PROGRAM PRG_Com
VAR
END_VAR

(*Instanitate Serial port com function *) 
//ChemRIXS PTM_03 
K2S17_E5_CH2_fbSerialLineControl(
	Mode:= SERIALLINEMODE_EL6_22B,
	pComIn:= ADR(K2S17_E5_CH2_stComIn),
	pComOut:=ADR(K2S17_E5_CH2_stComOut),
	SizeComIn:= SIZEOF(K2S17_E5_CH2_stComOut),
	TxBuffer:= K2S17_E5_CH2_SerialTXBuffer,
	RxBuffer:= K2S17_E5_CH2_SerialRXBuffer,
	Error=> ,
	ErrorID=> );
	
//ChemRIXS PTM_04
K2S17_E5_CH1_fbSerialLineControl(
	Mode:= SERIALLINEMODE_EL6_22B,
	pComIn:= ADR(K2S17_E5_CH1_stComIn),
	pComOut:=ADR(K2S17_E5_CH1_stComOut),
	SizeComIn:= SIZEOF(K2S17_E5_CH1_stComOut),
	TxBuffer:= K2S17_E5_CH1_SerialTXBuffer,
	RxBuffer:= K2S17_E5_CH1_SerialRXBuffer,
	Error=> ,
	ErrorID=> );

END_PROGRAM

(* stored: Version 1.1.0.1, ProductVersion 3.1.4022.18
   POU PRG_Com: Id {f62942d6-44b0-4dbc-ab5c-ec4f30fb3bd9}, SpecialFunc None *)
